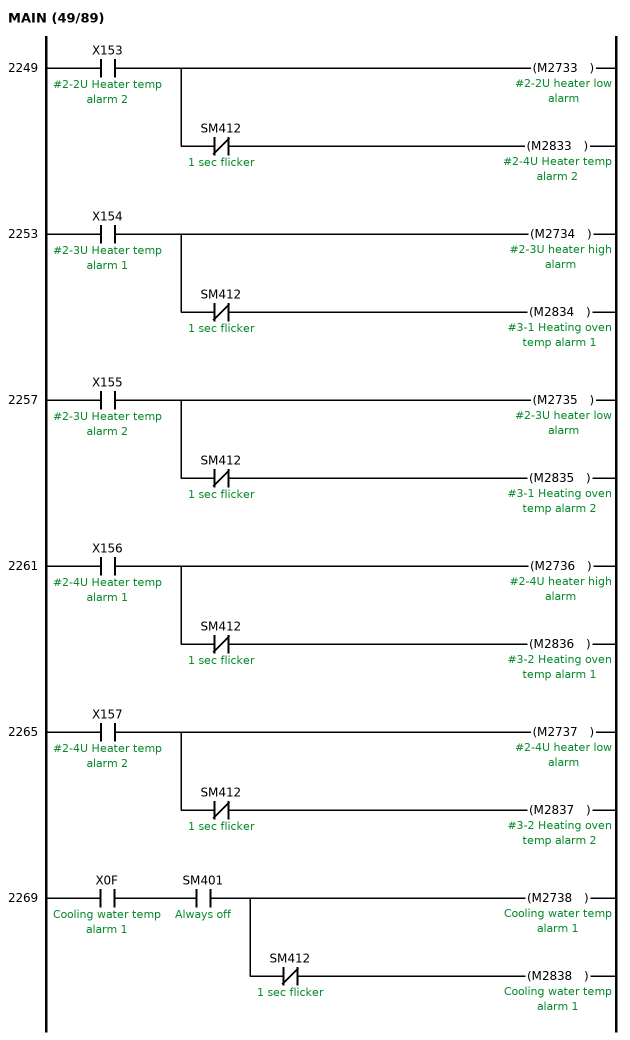
[picture p48: ladder of MAIN, rungs at steps 2249 to 2269]
2249  LD      X153  ; #2-2U Heater temp alarm 2
      OUT     M2733  ; #2-2U heater low alarm
      ANI     SM412  ; 1 sec flicker
      OUT     M2833  ; #2-4U Heater temp alarm 2
2253  LD      X154  ; #2-3U Heater temp alarm 1
      OUT     M2734  ; #2-3U heater high alarm
      ANI     SM412  ; 1 sec flicker
      OUT     M2834  ; #3-1 Heating oven temp alarm 1
2257  LD      X155  ; #2-3U Heater temp alarm 2
      OUT     M2735  ; #2-3U heater low alarm
      ANI     SM412  ; 1 sec flicker
      OUT     M2835  ; #3-1 Heating oven temp alarm 2
2261  LD      X156  ; #2-4U Heater temp alarm 1
      OUT     M2736  ; #2-4U heater high alarm
      ANI     SM412  ; 1 sec flicker
      OUT     M2836  ; #3-2 Heating oven temp alarm 1
2265  LD      X157  ; #2-4U Heater temp alarm 2
      OUT     M2737  ; #2-4U heater low alarm
      ANI     SM412  ; 1 sec flicker
      OUT     M2837  ; #3-2 Heating oven temp alarm 2
2269  LD      X0F  ; Cooling water temp alarm 1
      AND     SM401  ; Always off
      OUT     M2738  ; Cooling water temp alarm 1
      ANI     SM412  ; 1 sec flicker
      OUT     M2838  ; Cooling water temp alarm 1
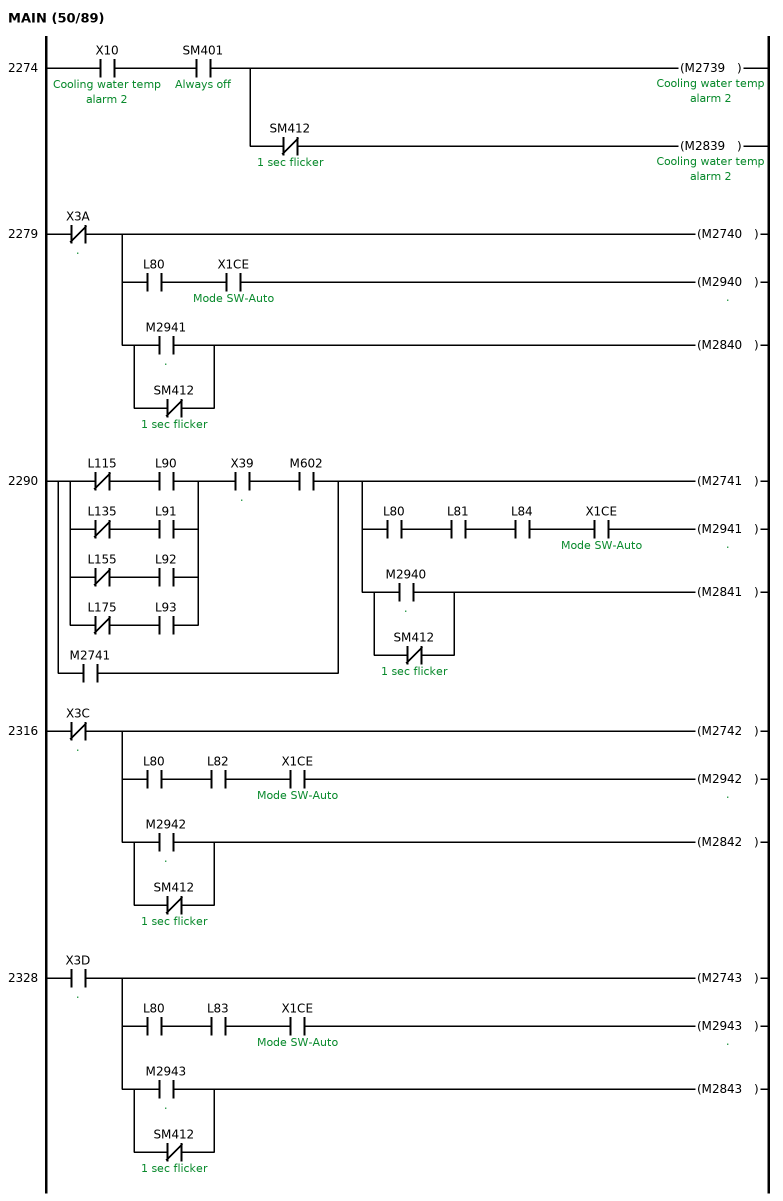
2274  LD      X10  ; Cooling water temp alarm 2
      AND     SM401  ; Always off
      OUT     M2739  ; Cooling water temp alarm 2
      ANI     SM412  ; 1 sec flicker
      OUT     M2839  ; Cooling water temp alarm 2
2279  LDI     X3A  ; .
      OUT     M2740
      MPS
      AND     L80
      AND     X1CE  ; Mode SW-Auto
      OUT     M2940  ; .
      MPP
      LD      M2941  ; .
      ORI     SM412  ; 1 sec flicker
      ANB
      OUT     M2840
2290  LDI     L115
      AND     L90
      LDI     L135
      AND     L91
      ORB
      LDI     L155
      AND     L92
      ORB
      LDI     L175
      AND     L93
      ORB
      AND     X39  ; .
      AND     M602
      OR      M2741
      OUT     M2741
      MPS
      AND     L80
      AND     L81
      AND     L84
      AND     X1CE  ; Mode SW-Auto
      OUT     M2941  ; .
      MPP
      LD      M2940  ; .
      ORI     SM412  ; 1 sec flicker
      ANB
      OUT     M2841
2316  LDI     X3C  ; .
      OUT     M2742
      MPS
      AND     L80
      AND     L82
      AND     X1CE  ; Mode SW-Auto
      OUT     M2942  ; .
      MPP
      LD      M2942  ; .
      ORI     SM412  ; 1 sec flicker
      ANB
      OUT     M2842
2328  LD      X3D  ; .
      OUT     M2743
      MPS
      AND     L80
      AND     L83
      AND     X1CE  ; Mode SW-Auto
      OUT     M2943  ; .
      MPP
      LD      M2943  ; .
      ORI     SM412  ; 1 sec flicker
      ANB
      OUT     M2843
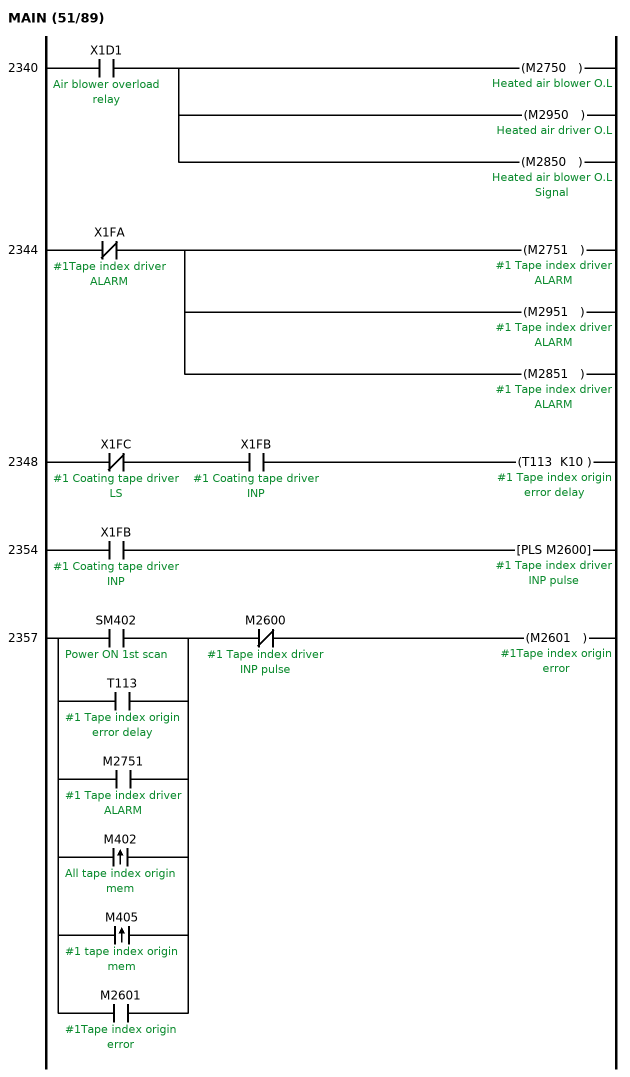
2340  LD      X1D1  ; Air blower overload relay
      OUT     M2750  ; Heated air blower O.L
      OUT     M2950  ; Heated air driver O.L
      OUT     M2850  ; Heated air blower O.L Signal
2344  LDI     X1FA  ; #1Tape index driver ALARM
      OUT     M2751  ; #1 Tape index driver ALARM
      OUT     M2951  ; #1 Tape index driver ALARM
      OUT     M2851  ; #1 Tape index driver ALARM
2348  LDI     X1FC  ; #1 Coating tape driver LS
      AND     X1FB  ; #1 Coating tape driver INP
      OUT     T113 K10  ; #1 Tape index origin error delay
2354  LD      X1FB  ; #1 Coating tape driver INP
      PLS     M2600  ; #1 Tape index driver INP pulse
2357  LD      SM402  ; Power ON 1st scan
      OR      T113  ; #1 Tape index origin error delay
      OR      M2751  ; #1 Tape index driver ALARM
      ORP     M402  ; All tape index origin mem
      ORP     M405  ; #1 tape index origin mem
      OR      M2601  ; #1Tape index origin error
      ANI     M2600  ; #1 Tape index driver INP pulse
      OUT     M2601  ; #1Tape index origin error
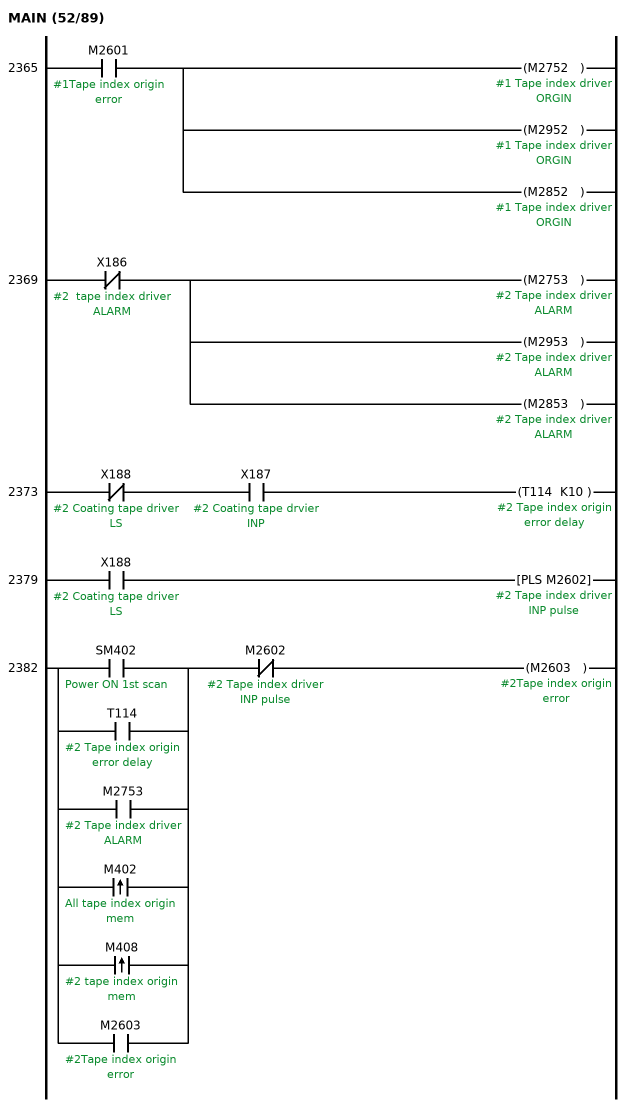
2365  LD      M2601  ; #1Tape index origin error
      OUT     M2752  ; #1 Tape index driver ORGIN
      OUT     M2952  ; #1 Tape index driver ORGIN
      OUT     M2852  ; #1 Tape index driver ORGIN
2369  LDI     X186  ; #2  tape index driver ALARM
      OUT     M2753  ; #2 Tape index driver ALARM
      OUT     M2953  ; #2 Tape index driver ALARM
      OUT     M2853  ; #2 Tape index driver ALARM
2373  LDI     X188  ; #2 Coating tape driver LS
      AND     X187  ; #2 Coating tape drvier INP
      OUT     T114 K10  ; #2 Tape index origin error delay
2379  LD      X188  ; #2 Coating tape driver LS
      PLS     M2602  ; #2 Tape index driver INP pulse
2382  LD      SM402  ; Power ON 1st scan
      OR      T114  ; #2 Tape index origin error delay
      OR      M2753  ; #2 Tape index driver ALARM
      ORP     M402  ; All tape index origin mem
      ORP     M408  ; #2 tape index origin mem
      OR      M2603  ; #2Tape index origin error
      ANI     M2602  ; #2 Tape index driver INP pulse
      OUT     M2603  ; #2Tape index origin error
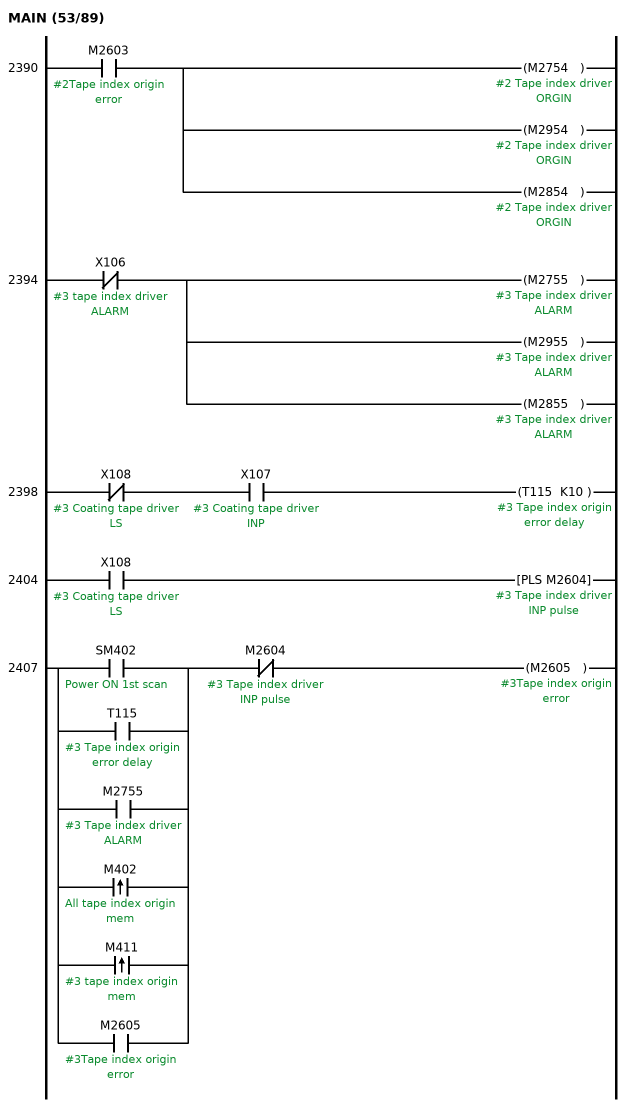
2390  LD      M2603  ; #2Tape index origin error
      OUT     M2754  ; #2 Tape index driver ORGIN
      OUT     M2954  ; #2 Tape index driver ORGIN
      OUT     M2854  ; #2 Tape index driver ORGIN
2394  LDI     X106  ; #3 tape index driver ALARM
      OUT     M2755  ; #3 Tape index driver ALARM
      OUT     M2955  ; #3 Tape index driver ALARM
      OUT     M2855  ; #3 Tape index driver ALARM
2398  LDI     X108  ; #3 Coating tape driver LS
      AND     X107  ; #3 Coating tape driver INP
      OUT     T115 K10  ; #3 Tape index origin error delay
2404  LD      X108  ; #3 Coating tape driver LS
      PLS     M2604  ; #3 Tape index driver INP pulse
2407  LD      SM402  ; Power ON 1st scan
      OR      T115  ; #3 Tape index origin error delay
      OR      M2755  ; #3 Tape index driver ALARM
      ORP     M402  ; All tape index origin mem
      ORP     M411  ; #3 tape index origin mem
      OR      M2605  ; #3Tape index origin error
      ANI     M2604  ; #3 Tape index driver INP pulse
      OUT     M2605  ; #3Tape index origin error
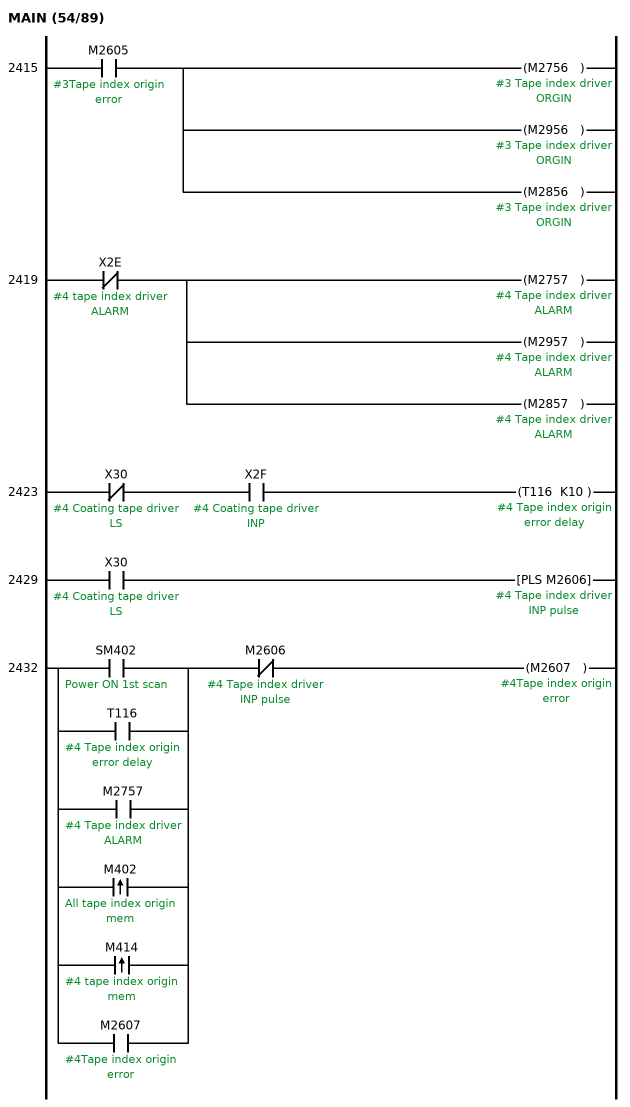
2415  LD      M2605  ; #3Tape index origin error
      OUT     M2756  ; #3 Tape index driver ORGIN
      OUT     M2956  ; #3 Tape index driver ORGIN
      OUT     M2856  ; #3 Tape index driver ORGIN
2419  LDI     X2E  ; #4 tape index driver ALARM
      OUT     M2757  ; #4 Tape index driver ALARM
      OUT     M2957  ; #4 Tape index driver ALARM
      OUT     M2857  ; #4 Tape index driver ALARM
2423  LDI     X30  ; #4 Coating tape driver LS
      AND     X2F  ; #4 Coating tape driver INP
      OUT     T116 K10  ; #4 Tape index origin error delay
2429  LD      X30  ; #4 Coating tape driver LS
      PLS     M2606  ; #4 Tape index driver INP pulse
2432  LD      SM402  ; Power ON 1st scan
      OR      T116  ; #4 Tape index origin error delay
      OR      M2757  ; #4 Tape index driver ALARM
      ORP     M402  ; All tape index origin mem
      ORP     M414  ; #4 tape index origin mem
      OR      M2607  ; #4Tape index origin error
      ANI     M2606  ; #4 Tape index driver INP pulse
      OUT     M2607  ; #4Tape index origin error
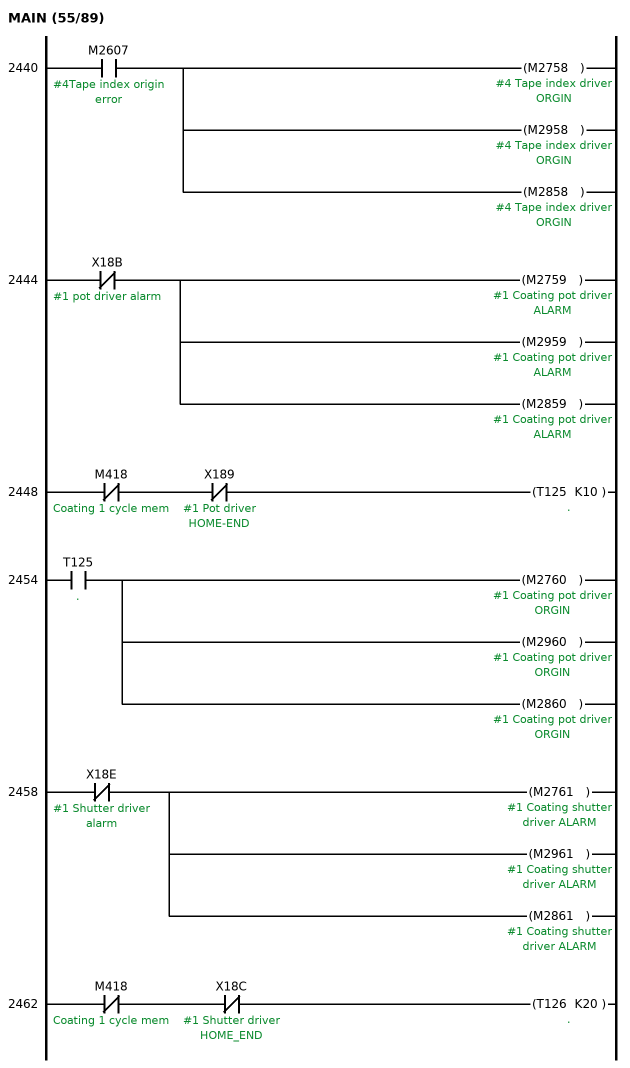
2440  LD      M2607  ; #4Tape index origin error
      OUT     M2758  ; #4 Tape index driver ORGIN
      OUT     M2958  ; #4 Tape index driver ORGIN
      OUT     M2858  ; #4 Tape index driver ORGIN
2444  LDI     X18B  ; #1 pot driver alarm
      OUT     M2759  ; #1 Coating pot driver ALARM
      OUT     M2959  ; #1 Coating pot driver ALARM
      OUT     M2859  ; #1 Coating pot driver ALARM
2448  LDI     M418  ; Coating 1 cycle mem
      ANI     X189  ; #1 Pot driver HOME-END
      OUT     T125 K10  ; .
2454  LD      T125  ; .
      OUT     M2760  ; #1 Coating pot driver ORGIN
      OUT     M2960  ; #1 Coating pot driver ORGIN
      OUT     M2860  ; #1 Coating pot driver ORGIN
2458  LDI     X18E  ; #1 Shutter driver alarm
      OUT     M2761  ; #1 Coating shutter driver ALARM
      OUT     M2961  ; #1 Coating shutter driver ALARM
      OUT     M2861  ; #1 Coating shutter driver ALARM
2462  LDI     M418  ; Coating 1 cycle mem
      ANI     X18C  ; #1 Shutter driver HOME_END
      OUT     T126 K20  ; .
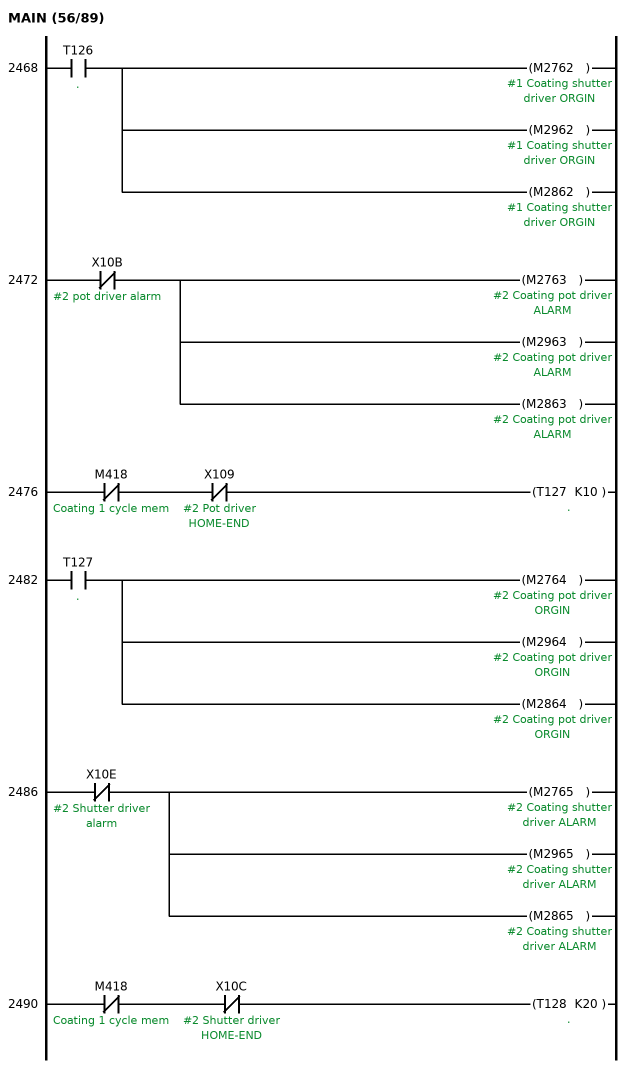
2468  LD      T126  ; .
      OUT     M2762  ; #1 Coating shutter driver ORGIN
      OUT     M2962  ; #1 Coating shutter driver ORGIN
      OUT     M2862  ; #1 Coating shutter driver ORGIN
2472  LDI     X10B  ; #2 pot driver alarm
      OUT     M2763  ; #2 Coating pot driver ALARM
      OUT     M2963  ; #2 Coating pot driver ALARM
      OUT     M2863  ; #2 Coating pot driver ALARM
2476  LDI     M418  ; Coating 1 cycle mem
      ANI     X109  ; #2 Pot driver HOME-END
      OUT     T127 K10  ; .
2482  LD      T127  ; .
      OUT     M2764  ; #2 Coating pot driver ORGIN
      OUT     M2964  ; #2 Coating pot driver ORGIN
      OUT     M2864  ; #2 Coating pot driver ORGIN
2486  LDI     X10E  ; #2 Shutter driver alarm
      OUT     M2765  ; #2 Coating shutter driver ALARM
      OUT     M2965  ; #2 Coating shutter driver ALARM
      OUT     M2865  ; #2 Coating shutter driver ALARM
2490  LDI     M418  ; Coating 1 cycle mem
      ANI     X10C  ; #2 Shutter driver HOME-END
      OUT     T128 K20  ; .
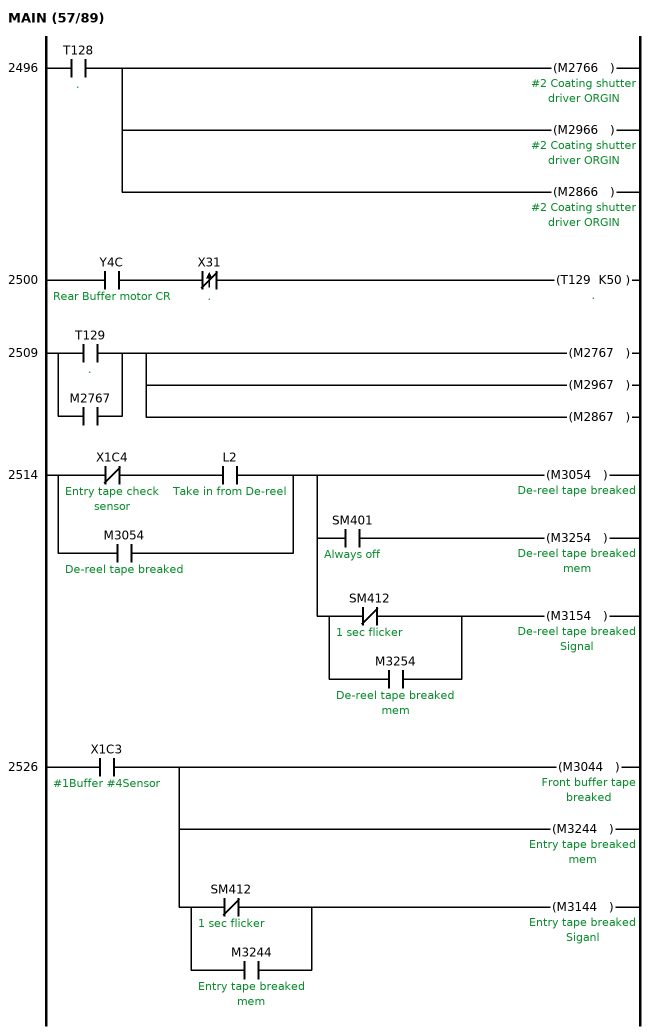
2496  LD      T128  ; .
      OUT     M2766  ; #2 Coating shutter driver ORGIN
      OUT     M2966  ; #2 Coating shutter driver ORGIN
      OUT     M2866  ; #2 Coating shutter driver ORGIN
2500  LD      Y4C  ; Rear Buffer motor CR
      ANDPI   X31  ; .
      OUT     T129 K50  ; .
2509  LD      T129  ; .
      OR      M2767
      OUT     M2767
      OUT     M2967
      OUT     M2867
2514  LDI     X1C4  ; Entry tape check sensor
      AND     L2  ; Take in from De-reel
      OR      M3054  ; De-reel tape breaked
      OUT     M3054  ; De-reel tape breaked
      MPS
      AND     SM401  ; Always off
      OUT     M3254  ; De-reel tape breaked mem
      MPP
      LDI     SM412  ; 1 sec flicker
      OR      M3254  ; De-reel tape breaked mem
      ANB
      OUT     M3154  ; De-reel tape breaked Signal
2526  LD      X1C3  ; #1Buffer #4Sensor
      OUT     M3044  ; Front buffer tape breaked
      OUT     M3244  ; Entry tape breaked mem
      LDI     SM412  ; 1 sec flicker
      OR      M3244  ; Entry tape breaked mem
      ANB
      OUT     M3144  ; Entry tape breaked Siganl
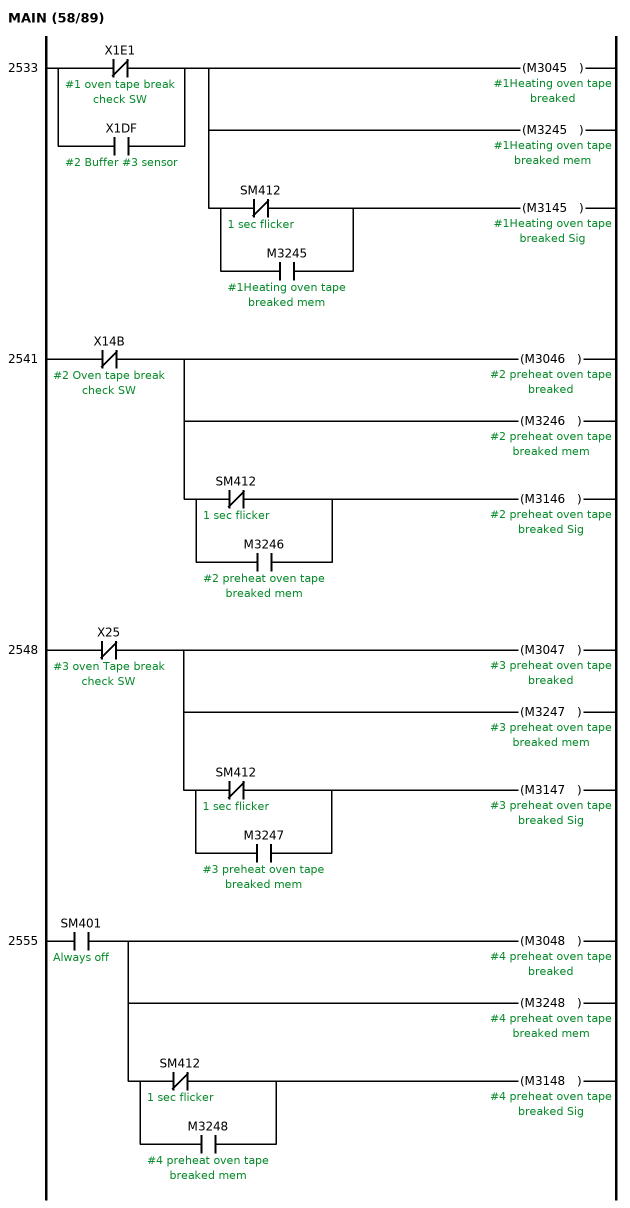
2533  LDI     X1E1  ; #1 oven tape break check SW
      OR      X1DF  ; #2 Buffer #3 sensor
      OUT     M3045  ; #1Heating oven tape breaked
      OUT     M3245  ; #1Heating oven tape breaked mem
      LDI     SM412  ; 1 sec flicker
      OR      M3245  ; #1Heating oven tape breaked mem
      ANB
      OUT     M3145  ; #1Heating oven tape breaked Sig
2541  LDI     X14B  ; #2 Oven tape break check SW
      OUT     M3046  ; #2 preheat oven tape breaked
      OUT     M3246  ; #2 preheat oven tape breaked mem
      LDI     SM412  ; 1 sec flicker
      OR      M3246  ; #2 preheat oven tape breaked mem
      ANB
      OUT     M3146  ; #2 preheat oven tape breaked Sig
2548  LDI     X25  ; #3 oven Tape break check SW
      OUT     M3047  ; #3 preheat oven tape breaked
      OUT     M3247  ; #3 preheat oven tape breaked mem
      LDI     SM412  ; 1 sec flicker
      OR      M3247  ; #3 preheat oven tape breaked mem
      ANB
      OUT     M3147  ; #3 preheat oven tape breaked Sig
2555  LD      SM401  ; Always off
      OUT     M3048  ; #4 preheat oven tape breaked
      OUT     M3248  ; #4 preheat oven tape breaked mem
      LDI     SM412  ; 1 sec flicker
      OR      M3248  ; #4 preheat oven tape breaked mem
      ANB
      OUT     M3148  ; #4 preheat oven tape breaked Sig
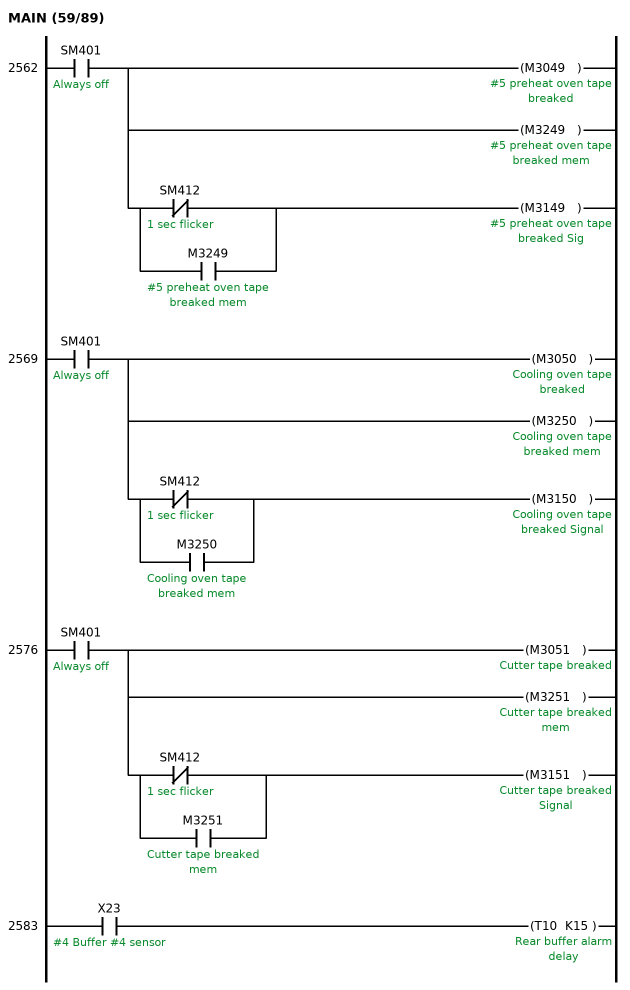
2562  LD      SM401  ; Always off
      OUT     M3049  ; #5 preheat oven tape breaked
      OUT     M3249  ; #5 preheat oven tape breaked mem
      LDI     SM412  ; 1 sec flicker
      OR      M3249  ; #5 preheat oven tape breaked mem
      ANB
      OUT     M3149  ; #5 preheat oven tape breaked Sig
2569  LD      SM401  ; Always off
      OUT     M3050  ; Cooling oven tape breaked
      OUT     M3250  ; Cooling oven tape breaked mem
      LDI     SM412  ; 1 sec flicker
      OR      M3250  ; Cooling oven tape breaked mem
      ANB
      OUT     M3150  ; Cooling oven tape breaked Signal
2576  LD      SM401  ; Always off
      OUT     M3051  ; Cutter tape breaked
      OUT     M3251  ; Cutter tape breaked mem
      LDI     SM412  ; 1 sec flicker
      OR      M3251  ; Cutter tape breaked mem
      ANB
      OUT     M3151  ; Cutter tape breaked Signal
2583  LD      X23  ; #4 Buffer #4 sensor
      OUT     T10 K15  ; Rear buffer alarm delay
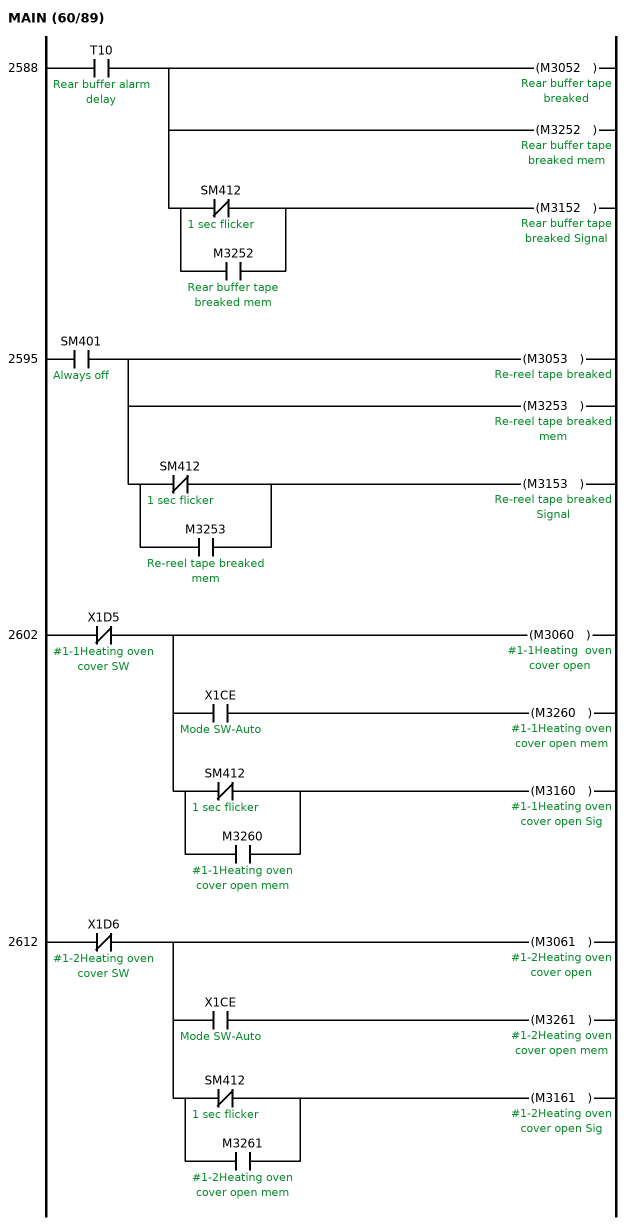
2588  LD      T10  ; Rear buffer alarm delay
      OUT     M3052  ; Rear buffer tape breaked
      OUT     M3252  ; Rear buffer tape breaked mem
      LDI     SM412  ; 1 sec flicker
      OR      M3252  ; Rear buffer tape breaked mem
      ANB
      OUT     M3152  ; Rear buffer tape breaked Signal
2595  LD      SM401  ; Always off
      OUT     M3053  ; Re-reel tape breaked
      OUT     M3253  ; Re-reel tape breaked mem
      LDI     SM412  ; 1 sec flicker
      OR      M3253  ; Re-reel tape breaked mem
      ANB
      OUT     M3153  ; Re-reel tape breaked Signal
2602  LDI     X1D5  ; #1-1Heating oven cover SW
      OUT     M3060  ; #1-1Heating  oven cover open
      MPS
      AND     X1CE  ; Mode SW-Auto
      OUT     M3260  ; #1-1Heating oven cover open mem
      MPP
      LDI     SM412  ; 1 sec flicker
      OR      M3260  ; #1-1Heating oven cover open mem
      ANB
      OUT     M3160  ; #1-1Heating oven cover open Sig
2612  LDI     X1D6  ; #1-2Heating oven cover SW
      OUT     M3061  ; #1-2Heating oven cover open
      MPS
      AND     X1CE  ; Mode SW-Auto
      OUT     M3261  ; #1-2Heating oven cover open mem
      MPP
      LDI     SM412  ; 1 sec flicker
      OR      M3261  ; #1-2Heating oven cover open mem
      ANB
      OUT     M3161  ; #1-2Heating oven cover open Sig
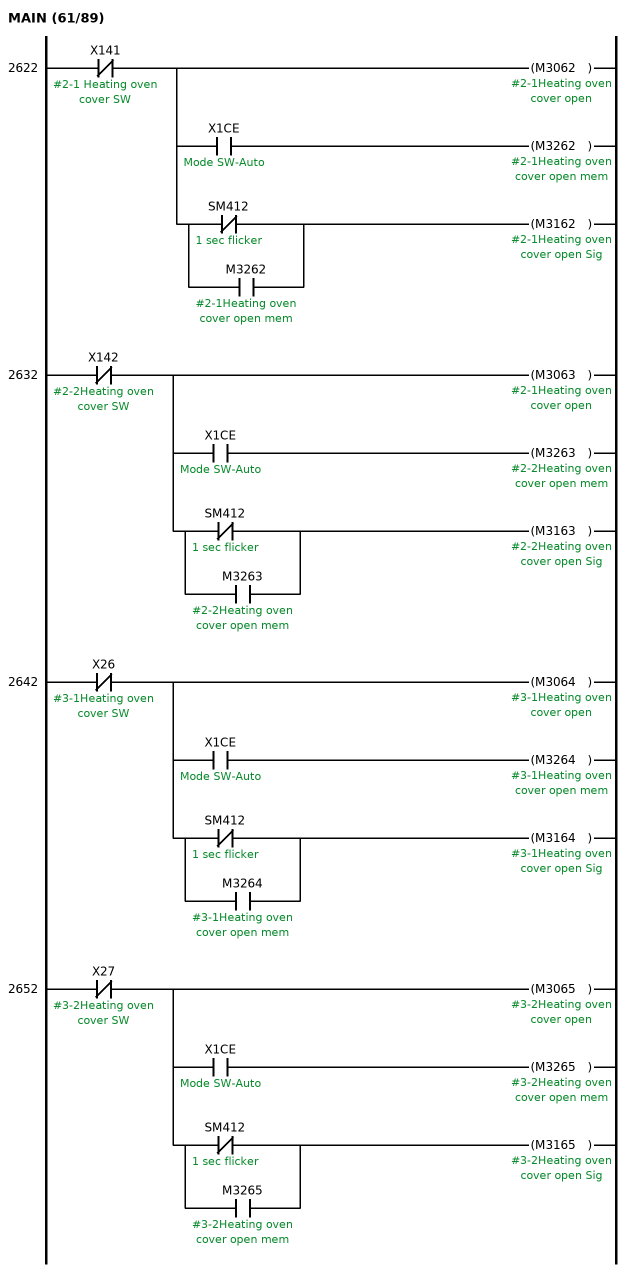
2622  LDI     X141  ; #2-1 Heating oven cover SW
      OUT     M3062  ; #2-1Heating oven cover open
      MPS
      AND     X1CE  ; Mode SW-Auto
      OUT     M3262  ; #2-1Heating oven cover open mem
      MPP
      LDI     SM412  ; 1 sec flicker
      OR      M3262  ; #2-1Heating oven cover open mem
      ANB
      OUT     M3162  ; #2-1Heating oven cover open Sig
2632  LDI     X142  ; #2-2Heating oven cover SW
      OUT     M3063  ; #2-1Heating oven cover open
      MPS
      AND     X1CE  ; Mode SW-Auto
      OUT     M3263  ; #2-2Heating oven cover open mem
      MPP
      LDI     SM412  ; 1 sec flicker
      OR      M3263  ; #2-2Heating oven cover open mem
      ANB
      OUT     M3163  ; #2-2Heating oven cover open Sig
2642  LDI     X26  ; #3-1Heating oven cover SW
      OUT     M3064  ; #3-1Heating oven cover open
      MPS
      AND     X1CE  ; Mode SW-Auto
      OUT     M3264  ; #3-1Heating oven cover open mem
      MPP
      LDI     SM412  ; 1 sec flicker
      OR      M3264  ; #3-1Heating oven cover open mem
      ANB
      OUT     M3164  ; #3-1Heating oven cover open Sig
2652  LDI     X27  ; #3-2Heating oven cover SW
      OUT     M3065  ; #3-2Heating oven cover open
      MPS
      AND     X1CE  ; Mode SW-Auto
      OUT     M3265  ; #3-2Heating oven cover open mem
      MPP
      LDI     SM412  ; 1 sec flicker
      OR      M3265  ; #3-2Heating oven cover open mem
      ANB
      OUT     M3165  ; #3-2Heating oven cover open Sig
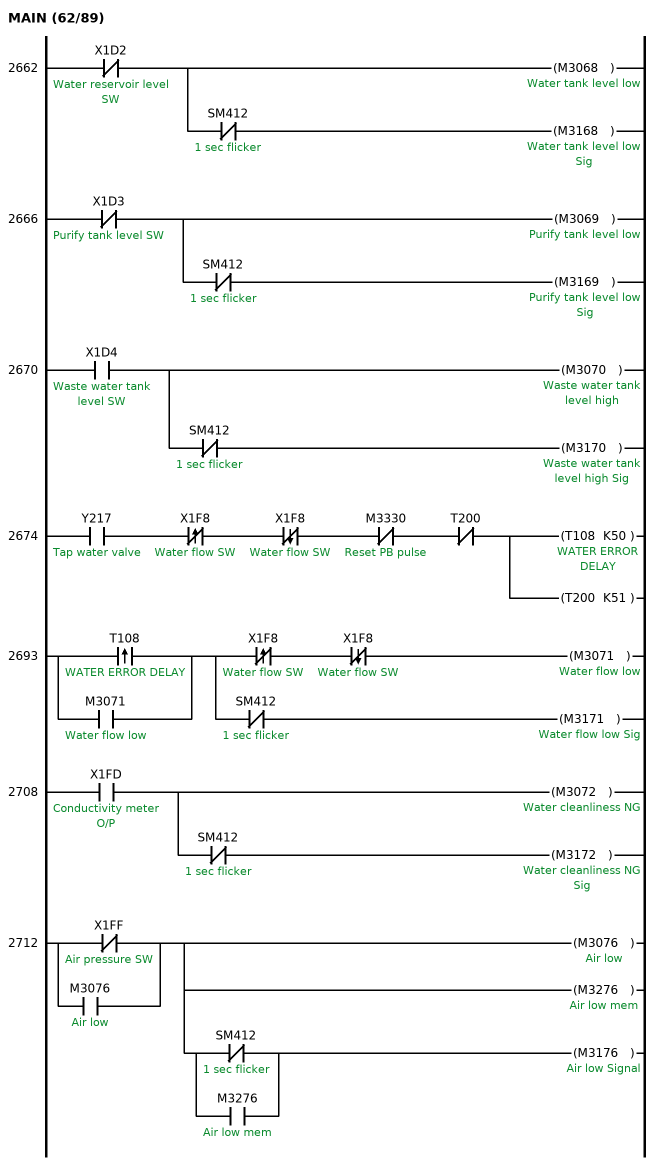
2662  LDI     X1D2  ; Water reservoir level SW
      OUT     M3068  ; Water tank level low
      ANI     SM412  ; 1 sec flicker
      OUT     M3168  ; Water tank level low Sig
2666  LDI     X1D3  ; Purify tank level SW
      OUT     M3069  ; Purify tank level low
      ANI     SM412  ; 1 sec flicker
      OUT     M3169  ; Purify tank level low Sig
2670  LD      X1D4  ; Waste water tank level SW
      OUT     M3070  ; Waste water tank level high
      ANI     SM412  ; 1 sec flicker
      OUT     M3170  ; Waste water tank level high Sig
2674  LD      Y217  ; Tap water valve
      ANDPI   X1F8  ; Water flow SW
      ANDFI   X1F8  ; Water flow SW
      ANI     M3330  ; Reset PB pulse
      ANI     T200
      OUT     T108 K50  ; WATER ERROR DELAY
      OUT     T200 K51
2693  LDP     T108  ; WATER ERROR DELAY
      OR      M3071  ; Water flow low
      MPS
      ANDPI   X1F8  ; Water flow SW
      ANDFI   X1F8  ; Water flow SW
      OUT     M3071  ; Water flow low
      MPP
      ANI     SM412  ; 1 sec flicker
      OUT     M3171  ; Water flow low Sig
2708  LD      X1FD  ; Conductivity meter O/P
      OUT     M3072  ; Water cleanliness NG
      ANI     SM412  ; 1 sec flicker
      OUT     M3172  ; Water cleanliness NG Sig
2712  LDI     X1FF  ; Air pressure SW
      OR      M3076  ; Air low
      OUT     M3076  ; Air low
      OUT     M3276  ; Air low mem
      LDI     SM412  ; 1 sec flicker
      OR      M3276  ; Air low mem
      ANB
      OUT     M3176  ; Air low Signal
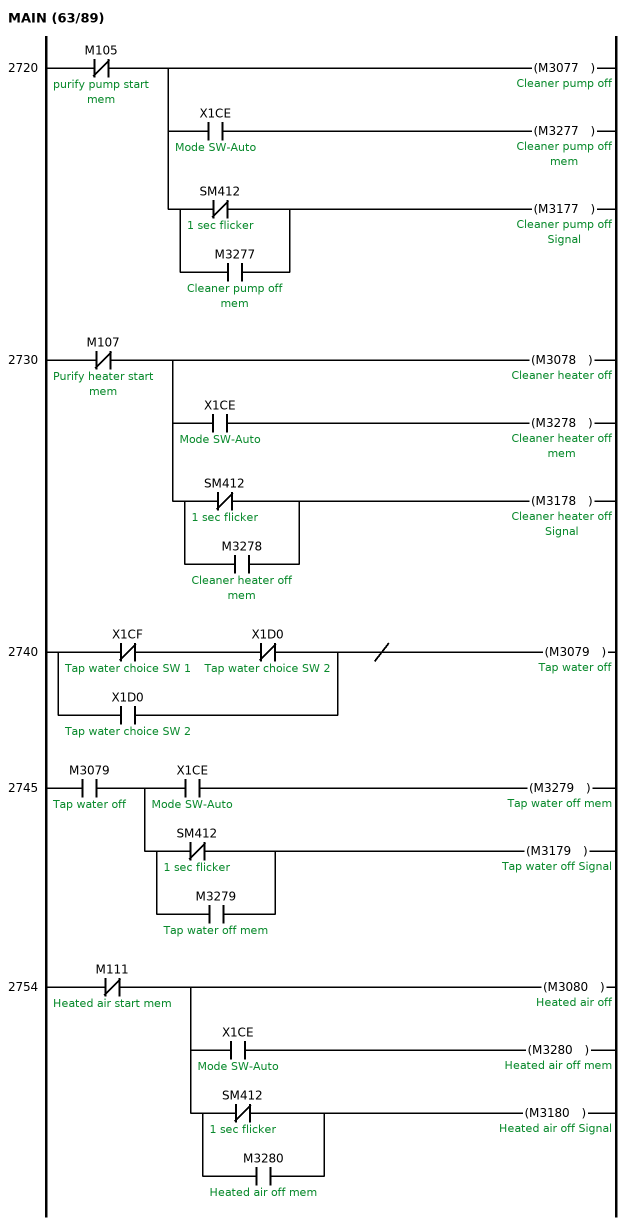
2720  LDI     M105  ; purify pump start mem
      OUT     M3077  ; Cleaner pump off
      MPS
      AND     X1CE  ; Mode SW-Auto
      OUT     M3277  ; Cleaner pump off mem
      MPP
      LDI     SM412  ; 1 sec flicker
      OR      M3277  ; Cleaner pump off mem
      ANB
      OUT     M3177  ; Cleaner pump off Signal
2730  LDI     M107  ; Purify heater start mem
      OUT     M3078  ; Cleaner heater off
      MPS
      AND     X1CE  ; Mode SW-Auto
      OUT     M3278  ; Cleaner heater off mem
      MPP
      LDI     SM412  ; 1 sec flicker
      OR      M3278  ; Cleaner heater off mem
      ANB
      OUT     M3178  ; Cleaner heater off Signal
2740  LDI     X1CF  ; Tap water choice SW 1
      ANI     X1D0  ; Tap water choice SW 2
      OR      X1D0  ; Tap water choice SW 2
      INV
      OUT     M3079  ; Tap water off
2745  LD      M3079  ; Tap water off
      MPS
      AND     X1CE  ; Mode SW-Auto
      OUT     M3279  ; Tap water off mem
      MPP
      LDI     SM412  ; 1 sec flicker
      OR      M3279  ; Tap water off mem
      ANB
      OUT     M3179  ; Tap water off Signal
2754  LDI     M111  ; Heated air start mem
      OUT     M3080  ; Heated air off
      MPS
      AND     X1CE  ; Mode SW-Auto
      OUT     M3280  ; Heated air off mem
      MPP
      LDI     SM412  ; 1 sec flicker
      OR      M3280  ; Heated air off mem
      ANB
      OUT     M3180  ; Heated air off Signal
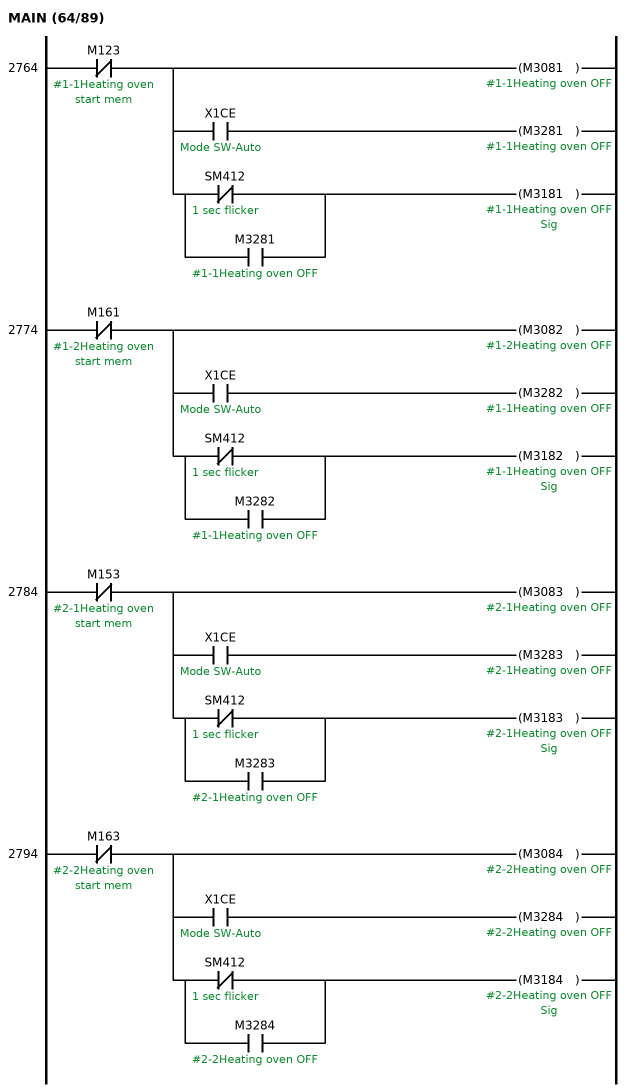
2764  LDI     M123  ; #1-1Heating oven start mem
      OUT     M3081  ; #1-1Heating oven OFF
      MPS
      AND     X1CE  ; Mode SW-Auto
      OUT     M3281  ; #1-1Heating oven OFF
      MPP
      LDI     SM412  ; 1 sec flicker
      OR      M3281  ; #1-1Heating oven OFF
      ANB
      OUT     M3181  ; #1-1Heating oven OFF Sig
2774  LDI     M161  ; #1-2Heating oven start mem
      OUT     M3082  ; #1-2Heating oven OFF
      MPS
      AND     X1CE  ; Mode SW-Auto
      OUT     M3282  ; #1-1Heating oven OFF
      MPP
      LDI     SM412  ; 1 sec flicker
      OR      M3282  ; #1-1Heating oven OFF
      ANB
      OUT     M3182  ; #1-1Heating oven OFF Sig
2784  LDI     M153  ; #2-1Heating oven start mem
      OUT     M3083  ; #2-1Heating oven OFF
      MPS
      AND     X1CE  ; Mode SW-Auto
      OUT     M3283  ; #2-1Heating oven OFF
      MPP
      LDI     SM412  ; 1 sec flicker
      OR      M3283  ; #2-1Heating oven OFF
      ANB
      OUT     M3183  ; #2-1Heating oven OFF Sig
2794  LDI     M163  ; #2-2Heating oven start mem
      OUT     M3084  ; #2-2Heating oven OFF
      MPS
      AND     X1CE  ; Mode SW-Auto
      OUT     M3284  ; #2-2Heating oven OFF
      MPP
      LDI     SM412  ; 1 sec flicker
      OR      M3284  ; #2-2Heating oven OFF
      ANB
      OUT     M3184  ; #2-2Heating oven OFF Sig
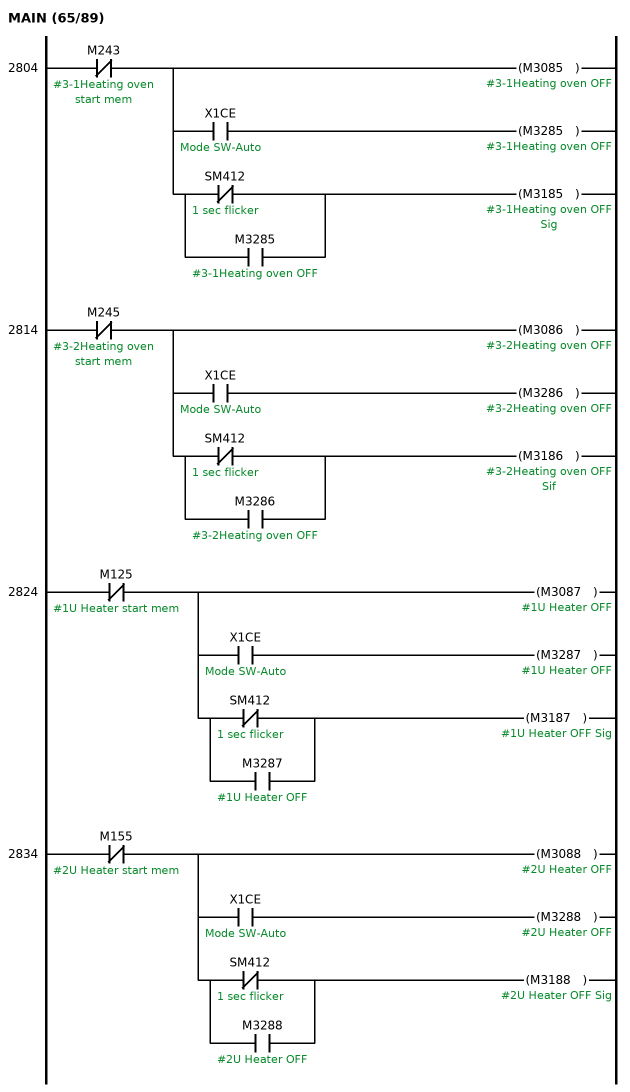
2804  LDI     M243  ; #3-1Heating oven start mem
      OUT     M3085  ; #3-1Heating oven OFF
      MPS
      AND     X1CE  ; Mode SW-Auto
      OUT     M3285  ; #3-1Heating oven OFF
      MPP
      LDI     SM412  ; 1 sec flicker
      OR      M3285  ; #3-1Heating oven OFF
      ANB
      OUT     M3185  ; #3-1Heating oven OFF Sig
2814  LDI     M245  ; #3-2Heating oven start mem
      OUT     M3086  ; #3-2Heating oven OFF
      MPS
      AND     X1CE  ; Mode SW-Auto
      OUT     M3286  ; #3-2Heating oven OFF
      MPP
      LDI     SM412  ; 1 sec flicker
      OR      M3286  ; #3-2Heating oven OFF
      ANB
      OUT     M3186  ; #3-2Heating oven OFF Sif
2824  LDI     M125  ; #1U Heater start mem
      OUT     M3087  ; #1U Heater OFF
      MPS
      AND     X1CE  ; Mode SW-Auto
      OUT     M3287  ; #1U Heater OFF
      MPP
      LDI     SM412  ; 1 sec flicker
      OR      M3287  ; #1U Heater OFF
      ANB
      OUT     M3187  ; #1U Heater OFF Sig
2834  LDI     M155  ; #2U Heater start mem
      OUT     M3088  ; #2U Heater OFF
      MPS
      AND     X1CE  ; Mode SW-Auto
      OUT     M3288  ; #2U Heater OFF
      MPP
      LDI     SM412  ; 1 sec flicker
      OR      M3288  ; #2U Heater OFF
      ANB
      OUT     M3188  ; #2U Heater OFF Sig
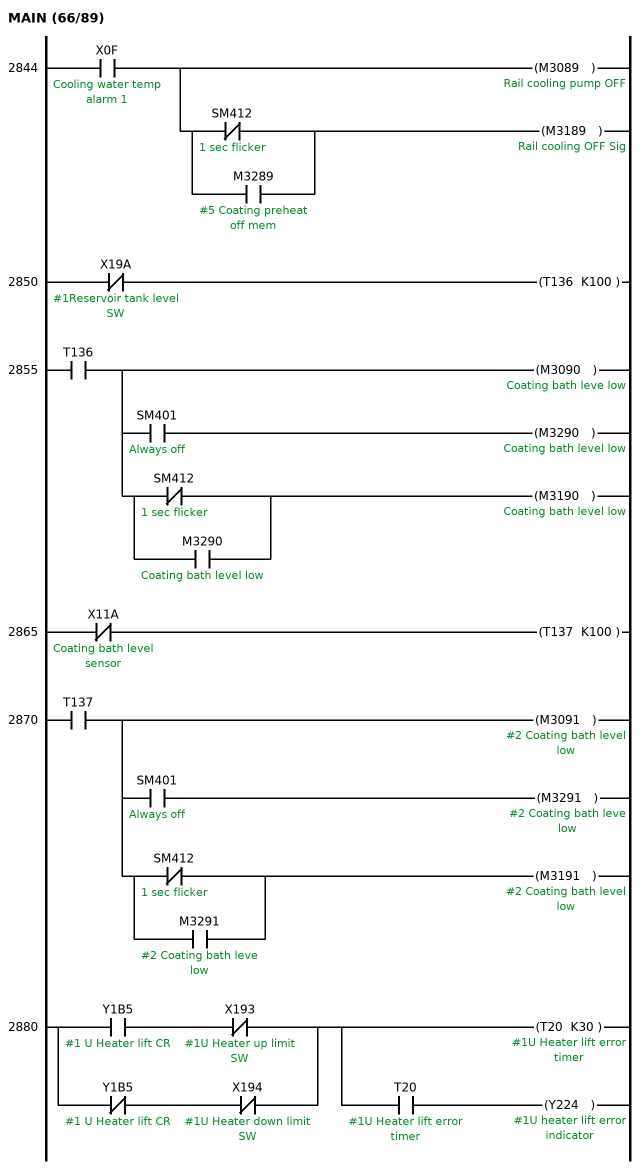
2844  LD      X0F  ; Cooling water temp alarm 1
      OUT     M3089  ; Rail cooling pump OFF
      LDI     SM412  ; 1 sec flicker
      OR      M3289  ; #5 Coating preheat off mem
      ANB
      OUT     M3189  ; Rail cooling OFF Sig
2850  LDI     X19A  ; #1Reservoir tank level SW
      OUT     T136 K100
2855  LD      T136
      OUT     M3090  ; Coating bath leve low
      MPS
      AND     SM401  ; Always off
      OUT     M3290  ; Coating bath level low
      MPP
      LDI     SM412  ; 1 sec flicker
      OR      M3290  ; Coating bath level low
      ANB
      OUT     M3190  ; Coating bath level low
2865  LDI     X11A  ; Coating bath level sensor
      OUT     T137 K100
2870  LD      T137
      OUT     M3091  ; #2 Coating bath level low
      MPS
      AND     SM401  ; Always off
      OUT     M3291  ; #2 Coating bath leve low
      MPP
      LDI     SM412  ; 1 sec flicker
      OR      M3291  ; #2 Coating bath leve low
      ANB
      OUT     M3191  ; #2 Coating bath level low
2880  LD      Y1B5  ; #1 U Heater lift CR
      ANI     X193  ; #1U Heater up limit SW
      LDI     Y1B5  ; #1 U Heater lift CR
      ANI     X194  ; #1U Heater down limit SW
      ORB
      OUT     T20 K30  ; #1U Heater lift error timer
      AND     T20  ; #1U Heater lift error timer
      OUT     Y224  ; #1U heater lift error indicator
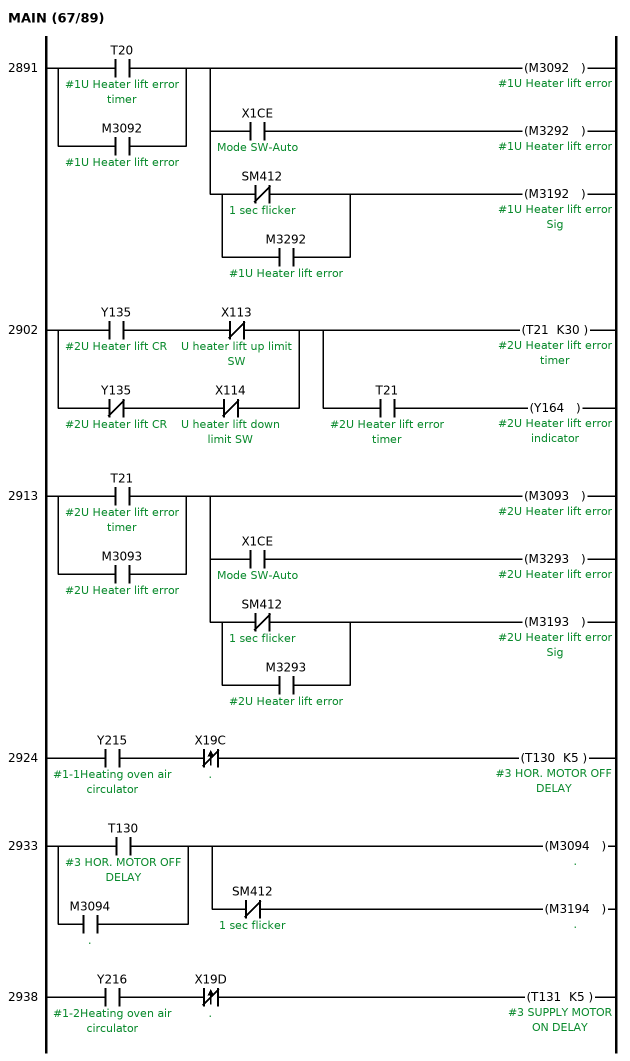
2891  LD      T20  ; #1U Heater lift error timer
      OR      M3092  ; #1U Heater lift error
      OUT     M3092  ; #1U Heater lift error
      MPS
      AND     X1CE  ; Mode SW-Auto
      OUT     M3292  ; #1U Heater lift error
      MPP
      LDI     SM412  ; 1 sec flicker
      OR      M3292  ; #1U Heater lift error
      ANB
      OUT     M3192  ; #1U Heater lift error Sig
2902  LD      Y135  ; #2U Heater lift CR
      ANI     X113  ; U heater lift up limit SW
      LDI     Y135  ; #2U Heater lift CR
      ANI     X114  ; U heater lift down limit SW
      ORB
      OUT     T21 K30  ; #2U Heater lift error timer
      AND     T21  ; #2U Heater lift error timer
      OUT     Y164  ; #2U Heater lift error indicator
2913  LD      T21  ; #2U Heater lift error timer
      OR      M3093  ; #2U Heater lift error
      OUT     M3093  ; #2U Heater lift error
      MPS
      AND     X1CE  ; Mode SW-Auto
      OUT     M3293  ; #2U Heater lift error
      MPP
      LDI     SM412  ; 1 sec flicker
      OR      M3293  ; #2U Heater lift error
      ANB
      OUT     M3193  ; #2U Heater lift error Sig
2924  LD      Y215  ; #1-1Heating oven air circulator
      ANDPI   X19C  ; .
      OUT     T130 K5  ; #3 HOR. MOTOR OFF DELAY
2933  LD      T130  ; #3 HOR. MOTOR OFF DELAY
      OR      M3094  ; .
      OUT     M3094  ; .
      ANI     SM412  ; 1 sec flicker
      OUT     M3194  ; .
2938  LD      Y216  ; #1-2Heating oven air circulator
      ANDPI   X19D  ; .
      OUT     T131 K5  ; #3 SUPPLY MOTOR ON DELAY
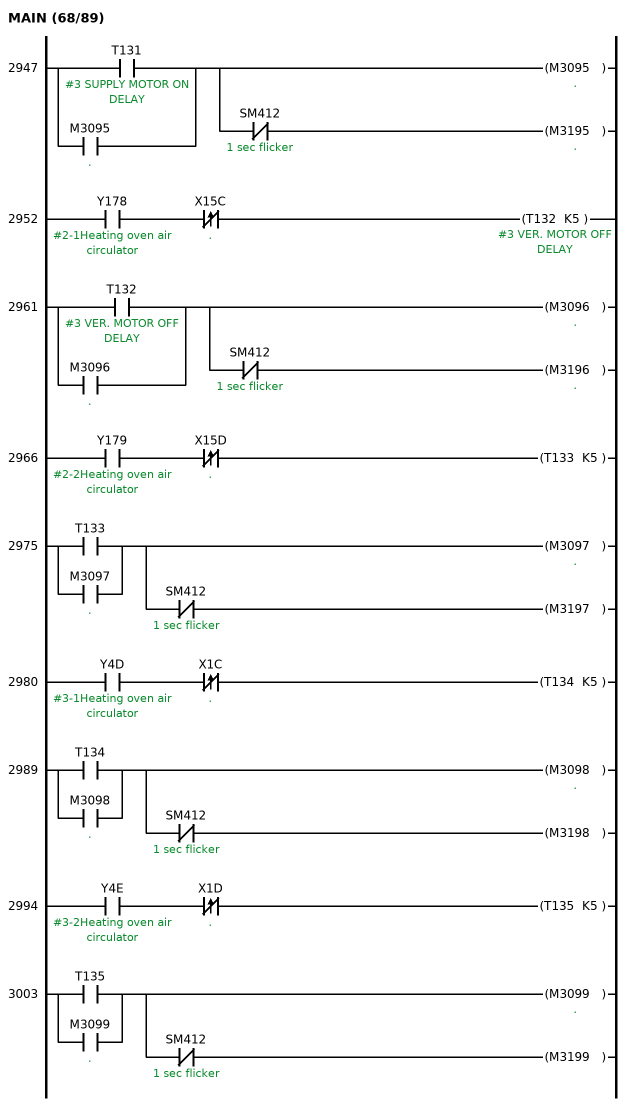
2947  LD      T131  ; #3 SUPPLY MOTOR ON DELAY
      OR      M3095  ; .
      OUT     M3095  ; .
      ANI     SM412  ; 1 sec flicker
      OUT     M3195  ; .
2952  LD      Y178  ; #2-1Heating oven air circulator
      ANDPI   X15C  ; .
      OUT     T132 K5  ; #3 VER. MOTOR OFF DELAY
2961  LD      T132  ; #3 VER. MOTOR OFF DELAY
      OR      M3096  ; .
      OUT     M3096  ; .
      ANI     SM412  ; 1 sec flicker
      OUT     M3196  ; .
2966  LD      Y179  ; #2-2Heating oven air circulator
      ANDPI   X15D  ; .
      OUT     T133 K5
2975  LD      T133
      OR      M3097  ; .
      OUT     M3097  ; .
      ANI     SM412  ; 1 sec flicker
      OUT     M3197
2980  LD      Y4D  ; #3-1Heating oven air circulator
      ANDPI   X1C  ; .
      OUT     T134 K5
2989  LD      T134
      OR      M3098  ; .
      OUT     M3098  ; .
      ANI     SM412  ; 1 sec flicker
      OUT     M3198
2994  LD      Y4E  ; #3-2Heating oven air circulator
      ANDPI   X1D  ; .
      OUT     T135 K5
3003  LD      T135
      OR      M3099  ; .
      OUT     M3099  ; .
      ANI     SM412  ; 1 sec flicker
      OUT     M3199
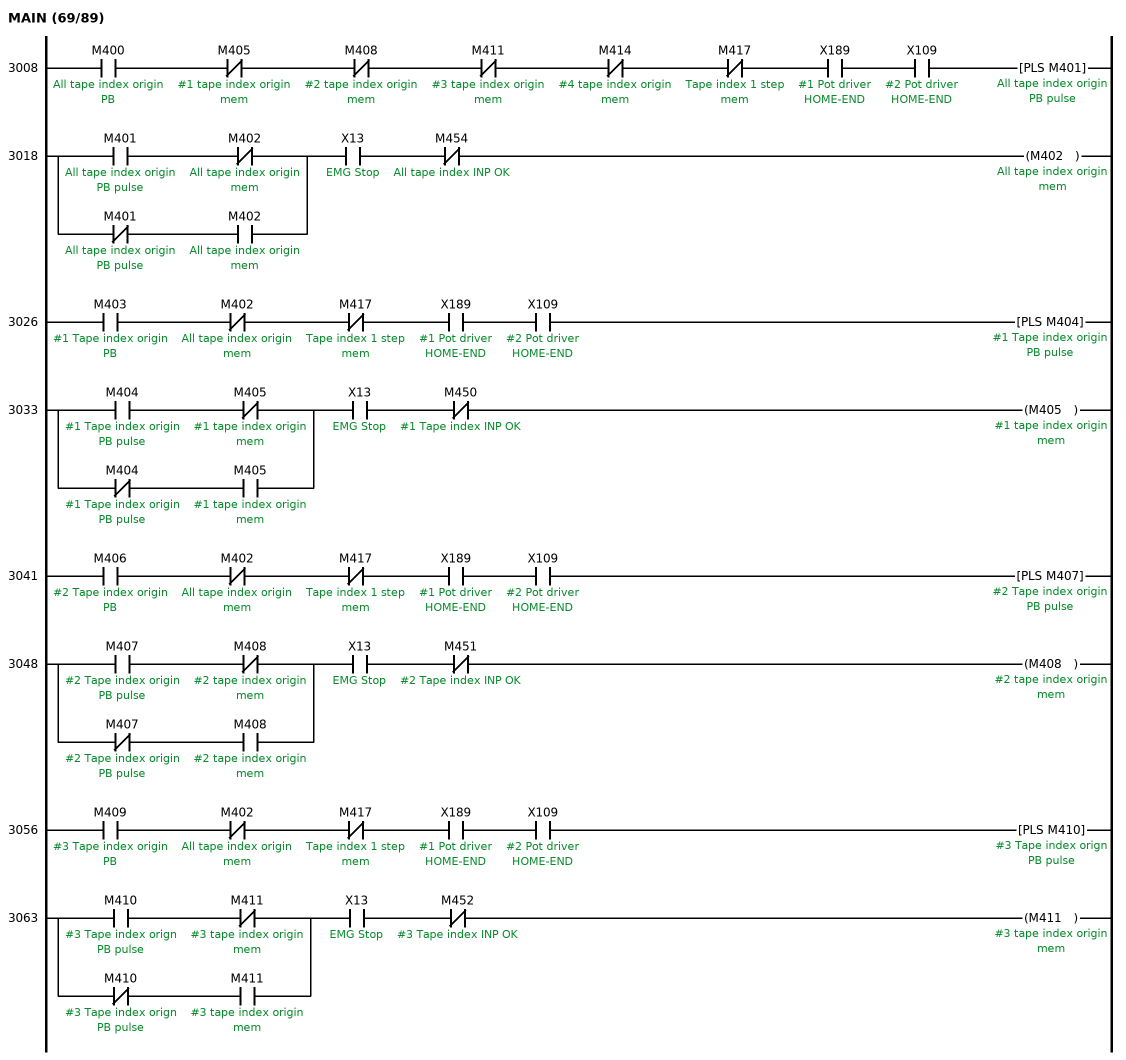
3008  LD      M400  ; All tape index origin PB
      ANI     M405  ; #1 tape index origin mem
      ANI     M408  ; #2 tape index origin mem
      ANI     M411  ; #3 tape index origin mem
      ANI     M414  ; #4 tape index origin mem
      ANI     M417  ; Tape index 1 step mem
      AND     X189  ; #1 Pot driver HOME-END
      AND     X109  ; #2 Pot driver HOME-END
      PLS     M401  ; All tape index origin PB pulse
3018  LD      M401  ; All tape index origin PB pulse
      ANI     M402  ; All tape index origin mem
      LDI     M401  ; All tape index origin PB pulse
      AND     M402  ; All tape index origin mem
      ORB
      AND     X13  ; EMG Stop
      ANI     M454  ; All tape index INP OK
      OUT     M402  ; All tape index origin mem
3026  LD      M403  ; #1 Tape index origin PB
      ANI     M402  ; All tape index origin mem
      ANI     M417  ; Tape index 1 step mem
      AND     X189  ; #1 Pot driver HOME-END
      AND     X109  ; #2 Pot driver HOME-END
      PLS     M404  ; #1 Tape index origin PB pulse
3033  LD      M404  ; #1 Tape index origin PB pulse
      ANI     M405  ; #1 tape index origin mem
      LDI     M404  ; #1 Tape index origin PB pulse
      AND     M405  ; #1 tape index origin mem
      ORB
      AND     X13  ; EMG Stop
      ANI     M450  ; #1 Tape index INP OK
      OUT     M405  ; #1 tape index origin mem
3041  LD      M406  ; #2 Tape index origin PB
      ANI     M402  ; All tape index origin mem
      ANI     M417  ; Tape index 1 step mem
      AND     X189  ; #1 Pot driver HOME-END
      AND     X109  ; #2 Pot driver HOME-END
      PLS     M407  ; #2 Tape index origin PB pulse
3048  LD      M407  ; #2 Tape index origin PB pulse
      ANI     M408  ; #2 tape index origin mem
      LDI     M407  ; #2 Tape index origin PB pulse
      AND     M408  ; #2 tape index origin mem
      ORB
      AND     X13  ; EMG Stop
      ANI     M451  ; #2 Tape index INP OK
      OUT     M408  ; #2 tape index origin mem
3056  LD      M409  ; #3 Tape index origin PB
      ANI     M402  ; All tape index origin mem
      ANI     M417  ; Tape index 1 step mem
      AND     X189  ; #1 Pot driver HOME-END
      AND     X109  ; #2 Pot driver HOME-END
      PLS     M410  ; #3 Tape index orign PB pulse
3063  LD      M410  ; #3 Tape index orign PB pulse
      ANI     M411  ; #3 tape index origin mem
      LDI     M410  ; #3 Tape index orign PB pulse
      AND     M411  ; #3 tape index origin mem
      ORB
      AND     X13  ; EMG Stop
      ANI     M452  ; #3 Tape index INP OK
      OUT     M411  ; #3 tape index origin mem
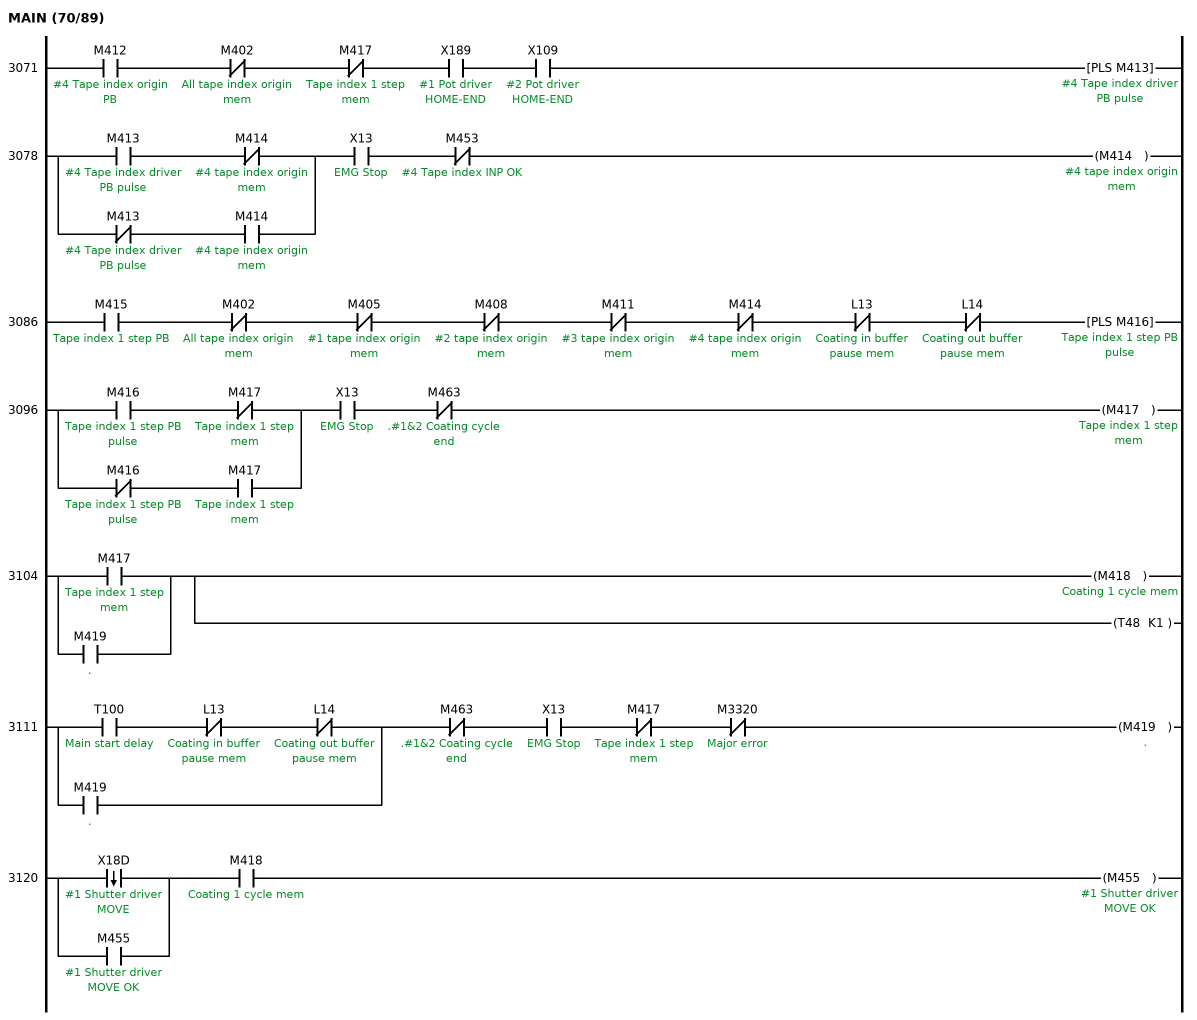
3071  LD      M412  ; #4 Tape index origin PB
      ANI     M402  ; All tape index origin mem
      ANI     M417  ; Tape index 1 step mem
      AND     X189  ; #1 Pot driver HOME-END
      AND     X109  ; #2 Pot driver HOME-END
      PLS     M413  ; #4 Tape index driver PB pulse
3078  LD      M413  ; #4 Tape index driver PB pulse
      ANI     M414  ; #4 tape index origin mem
      LDI     M413  ; #4 Tape index driver PB pulse
      AND     M414  ; #4 tape index origin mem
      ORB
      AND     X13  ; EMG Stop
      ANI     M453  ; #4 Tape index INP OK
      OUT     M414  ; #4 tape index origin mem
3086  LD      M415  ; Tape index 1 step PB
      ANI     M402  ; All tape index origin mem
      ANI     M405  ; #1 tape index origin mem
      ANI     M408  ; #2 tape index origin mem
      ANI     M411  ; #3 tape index origin mem
      ANI     M414  ; #4 tape index origin mem
      ANI     L13  ; Coating in buffer pause mem
      ANI     L14  ; Coating out buffer pause mem
      PLS     M416  ; Tape index 1 step PB pulse
3096  LD      M416  ; Tape index 1 step PB pulse
      ANI     M417  ; Tape index 1 step mem
      LDI     M416  ; Tape index 1 step PB pulse
      AND     M417  ; Tape index 1 step mem
      ORB
      AND     X13  ; EMG Stop
      ANI     M463  ; .#1&2 Coating cycle end
      OUT     M417  ; Tape index 1 step mem
3104  LD      M417  ; Tape index 1 step mem
      OR      M419  ; .
      OUT     M418  ; Coating 1 cycle mem
      OUT     T48 K1
3111  LD      T100  ; Main start delay
      ANI     L13  ; Coating in buffer pause mem
      ANI     L14  ; Coating out buffer pause mem
      OR      M419  ; .
      ANI     M463  ; .#1&2 Coating cycle end
      AND     X13  ; EMG Stop
      ANI     M417  ; Tape index 1 step mem
      ANI     M3320  ; Major error
      OUT     M419  ; .
3120  LDF     X18D  ; #1 Shutter driver MOVE
      OR      M455  ; #1 Shutter driver MOVE OK
      AND     M418  ; Coating 1 cycle mem
      OUT     M455  ; #1 Shutter driver MOVE OK
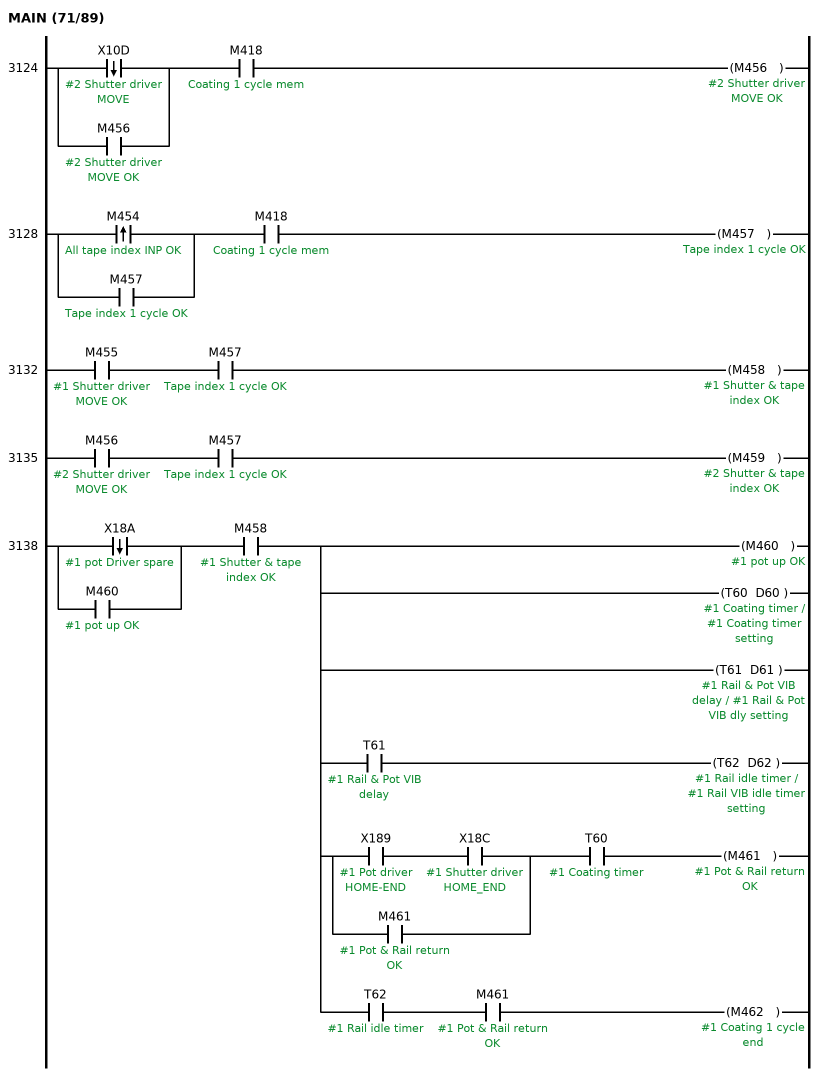
3124  LDF     X10D  ; #2 Shutter driver MOVE
      OR      M456  ; #2 Shutter driver MOVE OK
      AND     M418  ; Coating 1 cycle mem
      OUT     M456  ; #2 Shutter driver MOVE OK
3128  LDP     M454  ; All tape index INP OK
      OR      M457  ; Tape index 1 cycle OK
      AND     M418  ; Coating 1 cycle mem
      OUT     M457  ; Tape index 1 cycle OK
3132  LD      M455  ; #1 Shutter driver MOVE OK
      AND     M457  ; Tape index 1 cycle OK
      OUT     M458  ; #1 Shutter & tape index OK
3135  LD      M456  ; #2 Shutter driver MOVE OK
      AND     M457  ; Tape index 1 cycle OK
      OUT     M459  ; #2 Shutter & tape index OK
3138  LDF     X18A  ; #1 pot Driver spare
      OR      M460  ; #1 pot up OK
      AND     M458  ; #1 Shutter & tape index OK
      OUT     M460  ; #1 pot up OK
      OUT     T60 D60  ; #1 Coating timer / #1 Coating timer setting
      OUT     T61 D61  ; #1 Rail & Pot VIB delay / #1 Rail & Pot VIB dly setting
      MPS
      AND     T61  ; #1 Rail & Pot VIB delay
      OUT     T62 D62  ; #1 Rail idle timer / #1 Rail VIB idle timer setting
      MRD
      LD      X189  ; #1 Pot driver HOME-END
      AND     X18C  ; #1 Shutter driver HOME_END
      OR      M461  ; #1 Pot & Rail return OK
      ANB
      AND     T60  ; #1 Coating timer
      OUT     M461  ; #1 Pot & Rail return OK
      MPP
      AND     T62  ; #1 Rail idle timer
      AND     M461  ; #1 Pot & Rail return OK
      OUT     M462  ; #1 Coating 1 cycle end
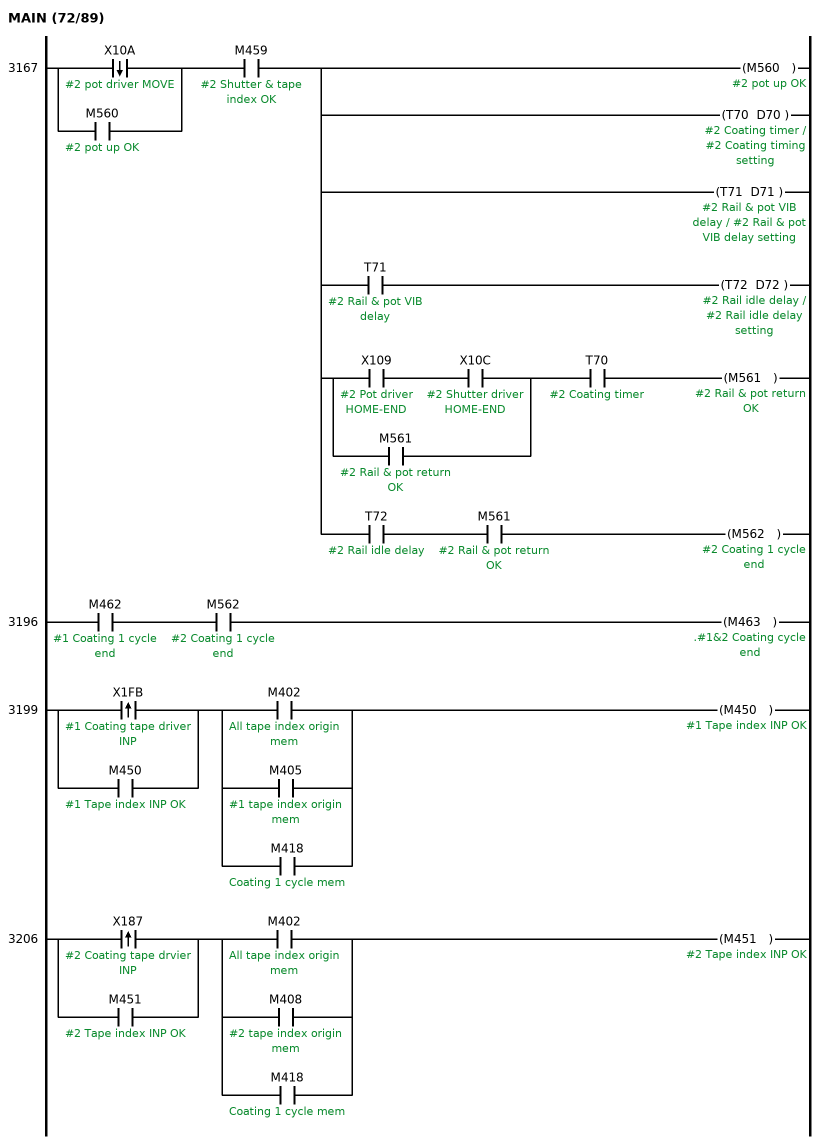
3167  LDF     X10A  ; #2 pot driver MOVE
      OR      M560  ; #2 pot up OK
      AND     M459  ; #2 Shutter & tape index OK
      OUT     M560  ; #2 pot up OK
      OUT     T70 D70  ; #2 Coating timer / #2 Coating timing setting
      OUT     T71 D71  ; #2 Rail & pot VIB delay / #2 Rail & pot VIB delay setting
      MPS
      AND     T71  ; #2 Rail & pot VIB delay
      OUT     T72 D72  ; #2 Rail idle delay / #2 Rail idle delay setting
      MRD
      LD      X109  ; #2 Pot driver HOME-END
      AND     X10C  ; #2 Shutter driver HOME-END
      OR      M561  ; #2 Rail & pot return OK
      ANB
      AND     T70  ; #2 Coating timer
      OUT     M561  ; #2 Rail & pot return OK
      MPP
      AND     T72  ; #2 Rail idle delay
      AND     M561  ; #2 Rail & pot return OK
      OUT     M562  ; #2 Coating 1 cycle end
3196  LD      M462  ; #1 Coating 1 cycle end
      AND     M562  ; #2 Coating 1 cycle end
      OUT     M463  ; .#1&2 Coating cycle end
3199  LDP     X1FB  ; #1 Coating tape driver INP
      OR      M450  ; #1 Tape index INP OK
      LD      M402  ; All tape index origin mem
      OR      M405  ; #1 tape index origin mem
      OR      M418  ; Coating 1 cycle mem
      ANB
      OUT     M450  ; #1 Tape index INP OK
3206  LDP     X187  ; #2 Coating tape drvier INP
      OR      M451  ; #2 Tape index INP OK
      LD      M402  ; All tape index origin mem
      OR      M408  ; #2 tape index origin mem
      OR      M418  ; Coating 1 cycle mem
      ANB
      OUT     M451  ; #2 Tape index INP OK
